KUKA KRL program: wkz2_an.src, wkz2_an.dat

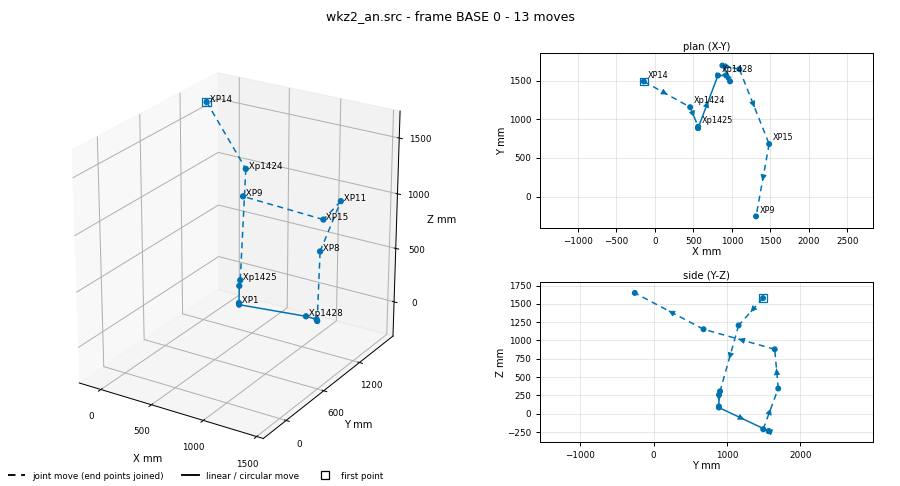
[picture p0: tool path of wkz2_an.src in frame BASE 0, 13 of 13 moves have a stored position in this frame; points joined in program order, loops and branches not executed]
--- wkz2_an.src ---
&ACCESS RVO2
&REL 308
&COMMENT Busca GUN X1
DEF wkz2_an( )
  ;FOLD INI;%{PE}%V2.2.2,%MKUKATPBASIS,%CINIT,%VCOMMON,%P
  ;FOLD BAS INI;%{PE}%V2.2.2,%MKUKATPBASIS,%CINIT,%VINIT,%P
  INTERRUPT DECL 3 WHEN $STOPMESS==TRUE DO IR_STOPM ( )
  INTERRUPT ON 3
  BAS (#INITMOV,0 )
  ;ENDFOLD
  ;FOLD A20 INI;%{E}%V2.2.2,%MKUKATPA20,%CINIT,%VINIT,%P
  IF ARC20==TRUE THEN
    A20 (ARC_INI)
    INTERRUPT DECL 6 WHEN $CYCFLAG[3]==FALSE DO A20(TECH_STOP2)
  ENDIF
  ;ENDFOLD
  ;FOLD A10 INI;%{E}%V2.2.2,%MKUKATPARC,%CINIT,%VINIT,%P
  IF A10_OPTION==#ACTIVE THEN
    INTERRUPT DECL 4 WHEN $CYCFLAG[2]==FALSE DO A10 (#APPL_ERROR)
    INTERRUPT DECL 7 WHEN A_ARC_SWI==#ACTIVE DO A10 (#ARC_SEAM)
    INTERRUPT DECL 5 WHEN A_FLY_ARC==TRUE DO A10 (#HPU_ARC)
    INTERRUPT  ON 5
    A10_INI ( )
  ENDIF
  ;ENDFOLD
  ;FOLD GRIPPER INI;%{E}%V2.2.2,%MKUKATPGRIPPER,%CINIT,%VINIT,%P
  USER_GRP(0,DUMMY,DUMMY,GDEFAULT)
  ;ENDFOLD
  ;FOLD TOUCHSENSE INI;%{E}%V2.2.2,%MKUKATPTS,%CINIT,%VINIT,%P
  IF H70_OPTION THEN
    INTERRUPT DECL 15 WHEN $MEAS_PULSE[TOUCH_I[TOUCH_ACTIVE].IN_NR] DO H70 (6,CD0 )
    INTERRUPT DECL 16 WHEN $ZERO_MOVE DO H70 (7,CD0 )
    INTERRUPT DECL 17 WHEN $TECHPAR_C[FG_TOUCH,8]>0.5 DO H70 (8,CD0)
    H70 (1,CD0 )
  ENDIF
  ;ENDFOLD
  ;FOLD USER INI;%{P}%V2.2.2,%MKUKATPUSER,%CINIT,%VINIT,%P
  ;Make your modifications here
  ;ENDFOLD
  ;ENDFOLD

; Caracterização dos meios de produção:
; Versão Atual:
; 19/07/2013 12:00 Name: P13.060-R3 CHANGES: Pega Pinça X1

chk_w8_wechs_ok ( )        ;VERIFICAÇÃO DE FERRAMENTA: toolchanger

;FOLD WAIT FOR IN 161 'deposito ocupado'  State= TRUE ;%{PE}%R 4.1.16,%MKUKATPBASIS,%CWAIT_FOR,%VWAIT_FOR,%P 1:0, 2:161, 3:'deposito ocupado', 5:TRUE, 6:
WAIT FOR $IN[161]==TRUE
;ENDFOLD
;FOLD WAIT FOR IN 219 'placas de suporte fundidas'  State= FALSE ;%{PE}%R 4.1.16,%MKUKATPBASIS,%CWAIT_FOR,%VWAIT_FOR,%P 1:0, 2:219, 3:'placas de suporte fundidas', 5:FALSE, 6:
WAIT FOR $IN[219]==FALSE
;ENDFOLD
;FOLD PULSE 167 'protecao da pinca abrir'  State= TRUE   Time= 3 sec;%{PE}%R 4.1.16,%MKUKATPBASIS,%COUT,%VPULSE,%P 2:167, 3:'protecao da pinca abrir', 5:TRUE, 6:, 8:3
PULSE($OUT[167], TRUE,3)
;ENDFOLD
;FOLD WAIT FOR IN 165 'protecao da pinca aberto'  State= TRUE ;%{PE}%R 4.1.16,%MKUKATPBASIS,%CWAIT_FOR,%VWAIT_FOR,%P 1:0, 2:165, 3:'protecao da pinca aberto', 5:TRUE, 6:
WAIT FOR $IN[165]==TRUE
;ENDFOLD

;FOLD PTP P14  Vel= 100 % PDAT13 Tool[8]:Tool Changer Base[0];%{PE}%R 4.1.16,%MKUKATPBASIS,%CMOVE,%VPTP,%P 1:PTP, 2:P14, 3:, 5:100, 7:PDAT13
$BWDSTART = FALSE
PDAT_ACT=PPDAT13
BAS(#PTP_DAT)
FDAT_ACT=FP14
BAS(#FRAMES)
BAS(#VEL_PTP,100)
PTP XP14
;ENDFOLD
;FOLD PTP p1424 CONT Vel= 100 % PDAT15 Tool[8]:Tool Changer Base[0];%{PE}%R 4.1.16,%MKUKATPBASIS,%CMOVE,%VPTP,%P 1:PTP, 2:p1424, 3:C_PTP, 5:100, 7:PDAT15
$BWDSTART = FALSE
PDAT_ACT=PPDAT15
BAS(#PTP_DAT)
FDAT_ACT=Fp1424
BAS(#FRAMES)
BAS(#VEL_PTP,100)
PTP Xp1424 C_PTP
;ENDFOLD

;FOLD OUT 224 'BLOQUEIA MPS'  State= FALSE ;%{PE}%R 4.1.16,%MKUKATPBASIS,%COUT,%VOUTX,%P 2:224, 3:'BLOQUEIA MPS', 5:FALSE, 6:
$OUT[224]=FALSE
;ENDFOLD
;FOLD OUT 223 'Desbloqueio MPS'  State= TRUE ;%{PE}%R 4.1.16,%MKUKATPBASIS,%COUT,%VOUTX,%P 2:223, 3:'Desbloqueio MPS', 5:TRUE, 6:
$OUT[223]=TRUE
;ENDFOLD

;FOLD PTP p1425 CONT Vel= 100 % PDAT16 Tool[8]:Tool Changer Base[0];%{PE}%R 4.1.16,%MKUKATPBASIS,%CMOVE,%VPTP,%P 1:PTP, 2:p1425, 3:C_PTP, 5:100, 7:PDAT16
$BWDSTART = FALSE
PDAT_ACT=PPDAT16
BAS(#PTP_DAT)
FDAT_ACT=Fp1425
BAS(#FRAMES)
BAS(#VEL_PTP,100)
PTP Xp1425 C_PTP
;ENDFOLD

;FOLD LIN p1426 CONT Vel= 0.3 m/s L_OLP1 Tool[8]:Tool Changer Base[0];%{PE}%R 4.1.16,%MKUKATPBASIS,%CMOVE,%VLIN,%P 1:LIN, 2:p1426, 3:C_DIS, 5:0.3, 7:L_OLP1
$BWDSTART = FALSE
LDAT_ACT=LL_OLP1
BAS(#CP_DAT)
FDAT_ACT=Fp1426
BAS(#FRAMES)
BAS(#VEL_CP,0.3)
LIN Xp1426 C_DIS
;ENDFOLD
;FOLD LIN P1 CONT Vel= 0.2 m/s CPDAT1 Tool[8]:Tool Changer Base[0];%{PE}%R 4.1.16,%MKUKATPBASIS,%CMOVE,%VLIN,%P 1:LIN, 2:P1, 3:C_DIS, 5:0.2, 7:CPDAT1
$BWDSTART = FALSE
LDAT_ACT=LCPDAT1
BAS(#CP_DAT)
FDAT_ACT=FP1
BAS(#FRAMES)
BAS(#VEL_CP,0.2)
LIN XP1 C_DIS
;ENDFOLD

;FOLD WAIT FOR IN 217 'MPS destravado'  State= TRUE ;%{PE}%R 4.1.16,%MKUKATPBASIS,%CWAIT_FOR,%VWAIT_FOR,%P 1:0, 2:217, 3:'MPS destravado', 5:TRUE, 6:
WAIT FOR $IN[217]==TRUE
;ENDFOLD
;FOLD WAIT FOR IN 221 'MPS travado'  State= FALSE ;%{PE}%R 4.1.16,%MKUKATPBASIS,%CWAIT_FOR,%VWAIT_FOR,%P 1:0, 2:221, 3:'MPS travado', 5:FALSE, 6:
WAIT FOR $IN[221]==FALSE
;ENDFOLD

;FOLD ; posicao de pega;%{PE}%R 4.1.16,%MKUKATPBASIS,%CCOMMENT,%VNORMAL,%P 2:posicao de pega
;ENDFOLD
;FOLD LIN p1427  Vel= 0.15 m/s L_OLP2 Tool[8]:Tool Changer Base[0];%{PE}%R 4.1.16,%MKUKATPBASIS,%CMOVE,%VLIN,%P 1:LIN, 2:p1427, 3:, 5:0.15, 7:L_OLP2
$BWDSTART = FALSE
LDAT_ACT=LL_OLP2
BAS(#CP_DAT)
FDAT_ACT=Fp1427
BAS(#FRAMES)
BAS(#VEL_CP,0.15)
LIN Xp1427
;ENDFOLD

;FOLD IBUS  OFF;%{PE}%R 4.1.16,%MKUKATPBASIS,%CIBUS,%VMAP,%P 2:#OFF, 3:1
$IBUS_OFF=$IBUS_ON
$IBUS_ON=0
;ENDFOLD
;FOLD OUT 223 'Desbloqueio MPS'  State= FALSE ;%{PE}%R 4.1.16,%MKUKATPBASIS,%COUT,%VOUTX,%P 2:223, 3:'Desbloqueio MPS', 5:FALSE, 6:
$OUT[223]=FALSE
;ENDFOLD
;FOLD OUT 224 'BLOQUEIA MPS'  State= TRUE ;%{PE}%R 4.1.16,%MKUKATPBASIS,%COUT,%VOUTX,%P 2:224, 3:'BLOQUEIA MPS', 5:TRUE, 6:
$OUT[224]=TRUE
;ENDFOLD
;FOLD WAIT FOR IN 219 'placas de suporte fundidas'  State= TRUE ;%{PE}%R 4.1.16,%MKUKATPBASIS,%CWAIT_FOR,%VWAIT_FOR,%P 1:0, 2:219, 3:'placas de suporte fundidas', 5:TRUE, 6:
WAIT FOR $IN[219]==TRUE
;ENDFOLD
;FOLD WAIT FOR IN 217 'MPS destravado'  State= FALSE ;%{PE}%R 4.1.16,%MKUKATPBASIS,%CWAIT_FOR,%VWAIT_FOR,%P 1:0, 2:217, 3:'MPS destravado', 5:FALSE, 6:
WAIT FOR $IN[217]==FALSE
;ENDFOLD
;FOLD WAIT FOR IN 221 'MPS travado'  State= TRUE ;%{PE}%R 4.1.16,%MKUKATPBASIS,%CWAIT_FOR,%VWAIT_FOR,%P 1:0, 2:221, 3:'MPS travado', 5:TRUE, 6:
WAIT FOR $IN[221]==TRUE
;ENDFOLD
;FOLD WAIT Time= 1 sec;%{PE}%R 4.1.16,%MKUKATPBASIS,%CWAIT,%VWAIT,%P 2:1
WAIT SEC 1
;ENDFOLD
;FOLD IBUS  ON SEGMENT_1;%{PE}%R 4.1.16,%MKUKATPBASIS,%CIBUS,%VMAP,%P 2:#ON, 3:1
$IBUS_ON=IBUS_SEGMENT[1]
$IBUS_OFF=0
;ENDFOLD
;FOLD WAIT Time= 2 sec;%{PE}%R 4.1.16,%MKUKATPBASIS,%CWAIT,%VWAIT,%P 2:2
WAIT SEC 2
;ENDFOLD

;FOLD ; saida com pinca;%{PE}%R 4.1.16,%MKUKATPBASIS,%CCOMMENT,%VNORMAL,%P 2:saida com pinca
;ENDFOLD
;FOLD LIN p1428  Vel= 0.2 m/s L_OLP3 Tool[2]:Gun X1                   Base[0];%{PE}%R 4.1.16,%MKUKATPBASIS,%CMOVE,%VLIN,%P 1:LIN, 2:p1428, 3:, 5:0.2, 7:L_OLP3
$BWDSTART = FALSE
LDAT_ACT=LL_OLP3
BAS(#CP_DAT)
FDAT_ACT=Fp1428
BAS(#FRAMES)
BAS(#VEL_CP,0.2)
LIN Xp1428
;ENDFOLD

;FOLD WAIT FOR IN 161 'deposito ocupado'  State= FALSE ;%{PE}%R 4.1.16,%MKUKATPBASIS,%CWAIT_FOR,%VWAIT_FOR,%P 1:0, 2:161, 3:'deposito ocupado', 5:FALSE, 6:
WAIT FOR $IN[161]==FALSE
;ENDFOLD
;FOLD WAIT FOR IN 219 'placas de suporte fundidas'  State= TRUE ;%{PE}%R 4.1.16,%MKUKATPBASIS,%CWAIT_FOR,%VWAIT_FOR,%P 1:0, 2:219, 3:'placas de suporte fundidas', 5:TRUE, 6:
WAIT FOR $IN[219]==TRUE
;ENDFOLD

;FOLD LIN P7 CONT Vel= 0.5 m/s CPDAT3 Tool[2]:Gun X1                   Base[0];%{PE}%R 4.1.16,%MKUKATPBASIS,%CMOVE,%VLIN,%P 1:LIN, 2:P7, 3:C_DIS, 5:0.5, 7:CPDAT3
$BWDSTART = FALSE
LDAT_ACT=LCPDAT3
BAS(#CP_DAT)
FDAT_ACT=FP7
BAS(#FRAMES)
BAS(#VEL_CP,0.5)
LIN XP7 C_DIS
;ENDFOLD

;FOLD PTP P13 CONT Vel= 100 % PDAT17 Tool[2]:Gun X1                   Base[0];%{PE}%R 4.1.16,%MKUKATPBASIS,%CMOVE,%VPTP,%P 1:PTP, 2:P13, 3:C_PTP, 5:100, 7:PDAT17
$BWDSTART = FALSE
PDAT_ACT=PPDAT17
BAS(#PTP_DAT)
FDAT_ACT=FP13
BAS(#FRAMES)
BAS(#VEL_PTP,100)
PTP XP13 C_PTP
;ENDFOLD
;FOLD PTP P8 CONT Vel= 100 % PDAT18 Tool[2]:Gun X1                   Base[0];%{PE}%R 4.1.16,%MKUKATPBASIS,%CMOVE,%VPTP,%P 1:PTP, 2:P8, 3:C_PTP, 5:100, 7:PDAT18
$BWDSTART = FALSE
PDAT_ACT=PPDAT18
BAS(#PTP_DAT)
FDAT_ACT=FP8
BAS(#FRAMES)
BAS(#VEL_PTP,100)
PTP XP8 C_PTP
;ENDFOLD
;FOLD PTP P11 CONT Vel= 100 % PDAT19 Tool[2]:Gun X1                   Base[0];%{PE}%R 4.1.16,%MKUKATPBASIS,%CMOVE,%VPTP,%P 1:PTP, 2:P11, 3:C_PTP, 5:100, 7:PDAT19
$BWDSTART = FALSE
PDAT_ACT=PPDAT19
BAS(#PTP_DAT)
FDAT_ACT=FP11
BAS(#FRAMES)
BAS(#VEL_PTP,100)
PTP XP11 C_PTP
;ENDFOLD
;FOLD PTP P15 CONT Vel= 100 % PDAT20 Tool[2]:Gun X1                   Base[0];%{PE}%R 4.1.16,%MKUKATPBASIS,%CMOVE,%VPTP,%P 1:PTP, 2:P15, 3:C_PTP, 5:100, 7:PDAT20
$BWDSTART = FALSE
PDAT_ACT=PPDAT20
BAS(#PTP_DAT)
FDAT_ACT=FP15
BAS(#FRAMES)
BAS(#VEL_PTP,100)
PTP XP15 C_PTP
;ENDFOLD
;FOLD PTP P9  Vel= 100 % PDAT7 Tool[2]:Gun X1                   Base[0];%{PE}%R 4.1.16,%MKUKATPBASIS,%CMOVE,%VPTP,%P 1:PTP, 2:P9, 3:, 5:100, 7:PDAT7
$BWDSTART = FALSE
PDAT_ACT=PPDAT7
BAS(#PTP_DAT)
FDAT_ACT=FP9
BAS(#FRAMES)
BAS(#VEL_PTP,100)
PTP XP9
;ENDFOLD

END

--- wkz2_an.dat ---
&ACCESS RVO2
&REL 308
&COMMENT Busca GUN X1
DEFDAT  WKZ2_AN
;FOLD EXTERNAL DECLARATIONS;%{PE}%V2.2.2,%MKUKATPBASIS,%CEXT,%VCOMMON,%P
;FOLD BAS EXT;%{PE}%V2.2.2,%MKUKATPBASIS,%CEXT,%VEXT,%P
EXT  BAS (BAS_COMMAND  :IN,REAL  :IN )
DECL INT SUCCESS
;ENDFOLD
;FOLD A10 EXT;%{E}%V2.2.2,%MKUKATPARC,%CEXT,%VEXT,%P
EXT  A10 (A_CMD_T  :IN,A_STRT_T  :IN,A_WELD_T  :IN,A_END_T  :IN,INT  :IN )
;ENDFOLD
;FOLD A20 EXT;%{E}%V2.2.2,%MKUKATPA20,%CEXT,%VEXT,%P
EXT  A20 (INT  :IN,WELD_ST  :IN,WELD_FI  :IN,INT  :IN )
;ENDFOLD
;FOLD GRIPPER EXT;%{E}%V2.2.2,%MKUKATPGRIPPER,%CEXT,%VEXT,%P
EXT  H50 (INT  :IN,INT  :IN,INT  :IN,GRP_TYP  :IN )
;ENDFOLD
;FOLD SPOT EXT;%{E}%V2.2.2,%MKUKATPSPOT,%CEXT,%VEXT,%P
EXT  USERSPOT (S_COMMAND  :IN,SPOT_TYPE  :IN )
;ENDFOLD
;FOLD TOUCHSENSE EXT;%{E}%V2.2.2,%MKUKATPTS,%CEXT,%VEXT,%P
EXT  H70 (INT  :IN,SRCH_TYP_2  :OUT,E6POS  :IN,SRCH_TYP_3  :IN,SRCH_TYP_2  :IN,SRCH_TYP_2  :IN,SRCH_TYP_2  :IN,SRCH_TYP_2  :IN,SRCH_TYP_2  :IN,INT  :IN )
;ENDFOLD
;FOLD USER EXT;%{}%V2.2.2,%MKUKATPUSER,%CEXT,%VEXT,%P
;Make here your modifications
;ENDFOLD
;ENDFOLD

;# ============ START PATH : zh_p13060r3_x1 =============
DECL FDAT Fp1424={TOOL_NO 8,BASE_NO 0,IPO_FRAME #BASE}
DECL PDAT PP_OLP1={VEL 100.0,ACC 85.0,APO_DIST 10.0}
DECL E6POS Xp1424={x 459.710388,y 1159.64197,z 1205.90698,a 6.99536991,b -18.3480091,c -156.822098,s 2,t 3,e1 0.0,e2 0.0,e3 0.0,e4 0.0,e5 0.0,e6 0.0}
DECL FDAT Fp1425={TOOL_NO 8,BASE_NO 0,IPO_FRAME #BASE}
DECL PDAT PP_OLP2={VEL 100.0,ACC 85.0,APO_DIST 5.0}
DECL E6POS Xp1425={x 563.29718,y 906.381775,z 306.939087,a -0.824041605,b 0.657010376,c 179.235596,s 6,t 19,e1 0.0,e2 0.0,e3 0.0,e4 0.0,e5 0.0,e6 0.0}
DECL FDAT Fp1426={TOOL_NO 8,BASE_NO 0,IPO_FRAME #BASE}
DECL E6POS Xp1426={x 562.583374,y 892.514282,z 259.609985,a -0.827672482,b 0.656243384,c 179.237701,s 2,t 11,e1 0.0,e2 0.0,e3 0.0,e4 0.0,e5 0.0,e6 0.0}
DECL LDAT LL_OLP1={VEL 0.25,ACC 100.0,APO_DIST 5.0,APO_FAC 0.0}
DECL FDAT Fp1427={TOOL_NO 8,BASE_NO 0,IPO_FRAME #BASE}
DECL E6POS Xp1427={x 562.79657,y 890.181396,z 85.2290573,a -0.731356025,b 0.510744393,c 179.514999,s 2,t 11,e1 0.0,e2 0.0,e3 0.0,e4 0.0,e5 0.0,e6 0.0}
DECL LDAT LL_OLP2={VEL 0.25,ACC 100.0,APO_DIST 0.0,APO_FAC 0.0}
DECL FDAT Fp1428={TOOL_NO 2,BASE_NO 0,IPO_FRAME #BASE}
DECL E6POS Xp1428={x 820.640198,y 1571.28699,z -236.615906,a 89.1448364,b 0.822555006,c 150.655701,s 2,t 11,e1 0.0,e2 0.0,e3 0.0,e4 0.0,e5 0.0,e6 0.0}
DECL LDAT LL_OLP3={VEL 0.25,ACC 95.0,APO_DIST 1.0,APO_FAC 0.0}
DECL E6POS XP1={x 560.723328,y 890.410217,z 100.439499,a -0.829497814,b 0.656647325,c 179.237,s 2,t 11,e1 0.0,e2 0.0,e3 0.0,e4 0.0,e5 0.0,e6 0.0}
DECL BASIS_SUGG_T LAST_BASIS={POINT1[] "P15                     ",POINT2[] "P15                     ",CP_PARAMS[] "CPDAT2                  ",PTP_PARAMS[] "PDAT14                  ",CONT[] "C_PTP                   ",CP_VEL[] "2                       ",PTP_VEL[] "100                     "}
DECL FDAT FP1={TOOL_NO 8,BASE_NO 0,IPO_FRAME #BASE}
DECL LDAT LCPDAT1={VEL 2.0,ACC 95.0,APO_DIST 2.0,APO_FAC 50.0}
DECL E6POS XP7={x 928.293213,y 1569.56799,z -237.756393,a 89.1427383,b 0.82290262,c 150.655502,s 2,t 11,e1 0.0,e2 0.0,e3 0.0,e4 0.0,e5 0.0,e6 0.0}
DECL FDAT FP7={TOOL_NO 2,BASE_NO 0,IPO_FRAME #BASE}
DECL E6POS XP8={x 877.505188,y 1700.41101,z 344.48111,a 95.1087418,b -10.5330801,c 159.930603,s 2,t 11,e1 0.0,e2 0.0,e3 0.0,e4 0.0,e5 0.0,e6 0.0}
DECL FDAT FP8={TOOL_NO 2,BASE_NO 0,IPO_FRAME #BASE}
DECL PDAT PPDAT6={VEL 100.0,ACC 85.0,APO_DIST 10.0}
DECL E6POS XP9={x 1314.83301,y -257.575897,z 1649.01099,a -78.0111389,b -26.3947792,c -156.342697,s 2,t 35,e1 0.0,e2 0.0,e3 0.0,e4 0.0,e5 0.0,e6 0.0}
DECL FDAT FP9={TOOL_NO 2,BASE_NO 0,IPO_FRAME #BASE}
DECL PDAT PPDAT7={VEL 100.0,ACC 100.0,APO_DIST 50.0}
DECL SPOT_SUGG_T LAST_SPOT={GUN[] "1                       ",RETR_CMD[] "#CLO                    ",CHOISE[] "#FIRST                  ",CLO_TM[] "1                       ",PGNO1[] "252                     ",PRESS1[] "0                       ",PGNO2[] "1                       ",PRESS2[] "0                       ",SPOT_PARAMS[] "NORMAL                  "}
DECL E6POS XP11={x 1098.51404,y 1652.521,z 880.444092,a 83.1566315,b -3.28524995,c 149.159698,s 2,t 11,e1 0.0,e2 0.0,e3 0.0,e4 0.0,e5 0.0,e6 0.0}
DECL FDAT FP11={TOOL_NO 2,BASE_NO 0,IPO_FRAME #BASE}
DECL PDAT PPDAT9={VEL 100.0,ACC 85.0,APO_DIST 10.0}
DECL LDAT LCPDAT3={VEL 2.0,ACC 100.0,APO_DIST 2.0,APO_FAC 50.0}
DECL E6POS XP13={x 977.22168,y 1494.84802,z -210.685104,a 89.6360016,b 7.16609907,c 156.886002,s 2,t 11,e1 0.0,e2 0.0,e3 0.0,e4 0.0,e5 0.0,e6 0.0}
DECL FDAT FP13={TOOL_NO 2,BASE_NO 0,IPO_FRAME #BASE}
DECL PDAT PPDAT12={VEL 100.0,ACC 85.0,APO_DIST 10.0}
DECL E6POS XP14={x -141.548706,y 1492.88196,z 1578.60596,a -66.2912827,b 36.3567505,c -163.568695,s 2,t 3,e1 0.0,e2 0.0,e3 0.0,e4 0.0,e5 0.0,e6 0.0}
DECL FDAT FP14={TOOL_NO 8,BASE_NO 0,IPO_FRAME #BASE}
DECL PDAT PPDAT13={VEL 100.0,ACC 100.0,APO_DIST 10.0}
DECL E6POS XP15={x 1484.77698,y 681.020081,z 1153.60596,a -5.02922297,b -17.7332306,c 156.413101,s 2,t 3,e1 0.0,e2 0.0,e3 0.0,e4 0.0,e5 0.0,e6 0.0}
DECL FDAT FP15={TOOL_NO 2,BASE_NO 0,IPO_FRAME #BASE}
DECL PDAT PPDAT14={VEL 100.0,ACC 100.0,APO_DIST 10.0}
DECL LDAT LCPDAT9={VEL 2.0,ACC 100.0,APO_DIST 100.0,APO_FAC 50.0}
DECL PDAT PPDAT15={VEL 100.0,ACC 100.0,APO_DIST 10.0}
DECL LDAT LCPDAT4={VEL 2.0,ACC 100.0,APO_DIST 100.0,APO_FAC 50.0}
DECL PDAT PPDAT16={VEL 100.0,ACC 100.0,APO_DIST 5.0}
DECL LDAT LCPDAT5={VEL 2.0,ACC 100.0,APO_DIST 100.0,APO_FAC 50.0}
DECL PDAT PPDAT17={VEL 100.0,ACC 100.0,APO_DIST 10.0}
DECL LDAT LCPDAT6={VEL 2.0,ACC 100.0,APO_DIST 100.0,APO_FAC 50.0}
DECL PDAT PPDAT18={VEL 100.0,ACC 100.0,APO_DIST 30.0}
DECL LDAT LCPDAT7={VEL 2.0,ACC 100.0,APO_DIST 100.0,APO_FAC 50.0}
DECL PDAT PPDAT19={VEL 100.0,ACC 100.0,APO_DIST 50.0}
DECL LDAT LCPDAT8={VEL 2.0,ACC 100.0,APO_DIST 100.0,APO_FAC 50.0}
DECL PDAT PPDAT20={VEL 100.0,ACC 100.0,APO_DIST 30.0}
ENDDAT
